PROGRAM MAIN
VAR
END_VAR

// unit tests
MobjectCollectionsUnitTests();
MobjectConvertersUnitTests();
MobjectDatatypesUnitTests();
MobjectDeserializationUnitTests();
MobjectDisposableUnitTests();
MobjectErrorsUnitTests();
MobjectEventsUnitTests();
MobjectJsonUnitTests();
MobjectServerUnitTests();

// examples
MobjectCollectionsExample();

// tcunit
TcUnit.RUN();

END_PROGRAM

(* stored: Version 1.1.0.1, ProductVersion 3.1.4026.13
   POU MAIN: Id {42ba3a90-05d7-0643-1254-d4b210024561}, SpecialFunc None *)
